FUNCTION_BLOCK Drill
  (* Standard: 61499-2 *)
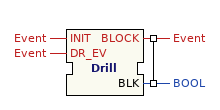
  EVENT_INPUT
    INIT;
    DR_EV;
  END_EVENT
  EVENT_OUTPUT
    BLOCK WITH BLK;
  END_EVENT
  VAR_OUTPUT
    BLK : BOOL;
  END_VAR
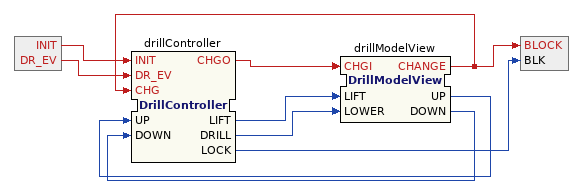
  FBS
    drillController : DrillController;
    drillModelView : DrillModelView;
  END_FBS
  EVENT_CONNECTIONS
    drillController.CHGO TO drillModelView.CHGI;
    INIT TO drillController.INIT;
    DR_EV TO drillController.DR_EV;
    drillModelView.CHANGE TO drillController.CHG;
    drillModelView.CHANGE TO BLOCK;
  END_CONNECTIONS
  DATA_CONNECTIONS
    drillController.LIFT TO drillModelView.LIFT;
    drillController.DRILL TO drillModelView.LOWER;
    drillModelView.UP TO drillController.UP;
    drillModelView.DOWN TO drillController.DOWN;
    drillController.LOCK TO BLK;
  END_CONNECTIONS
END_FUNCTION_BLOCK
